FUNCTION_BLOCK NodeFactory_Literal_BOOL EXTENDS NodeFactory

METHOD PUBLIC Create : I_Node
VAR
	pointerToNode : POINTER TO Node_Literal_BOOL;
END_VAR
pointerToNode := __NEW(Node_Literal_BOOL);
Create := pointerToNode^;
END_METHOD

END_FUNCTION_BLOCK

(* stored: Version 1.1.0.1, ProductVersion 3.1.4024.12
   POU NodeFactory_Literal_BOOL: Id {40e820c9-6ab1-083f-1936-ca01744bb371}, SpecialFunc None
   Method Create: Id {3a6095c4-583b-025f-0bfd-409922db5993} *)
